TYPE ST_SafetyOutput :
STRUCT
	abLinkedAxes : ARRAY[1..GVL_APP.nAXIS_NUM] OF BOOL; //boolean array for all axes
	sName : STRING; //Name descriptor for the safety output
	bTripped : BOOL;
	iSafetyOutputGroup : INT;
	
	//Correct terminology? What else is needed?
END_STRUCT
END_TYPE

(* stored: Version 1.1.0.1, ProductVersion 3.1.4024.11
   DUT ST_SafetyOutput: Id {8a85b2a5-61fa-4f89-9d55-2acad09a8c3a} *)
